TYPE
    ST_MyComponent_Status_1 : STRUCT
        Extended   : BOOL;
        Retracted  : BOOL;
        Extending  : BOOL;
        Retracting : BOOL;
    END_STRUCT
END_TYPE

(* stored: Version 1.1.0.1
   DUT ST_MyComponent_Status_1: Id {d433b09c-ab7b-4e77-9029-804e9da9f494} *)
